PROGRAM PRG_LVCP5_Group1
VAR
    // Function Block Instance
    fbContactor: FB_ContactorControl;

    // Contactor 1 IO Structure  
    stContactor_IO: ST_ContactorIO;
    
    // Başlangıç konfigürasyonu için flag
    bContactorInitDone: BOOL := FALSE;
    bCapacitorInitDone: BOOL := FALSE;	
END_VAR



	M_Contactor();
	
	M_Capacitor();

METHOD M_Capacitor : BOOL
VAR
    nGroupIndex : INT;
END_VAR
	nGroupIndex := 0;  // Grup 1 için index
	
	IF NOT bCapacitorInitDone THEN
	
		// Grup 1 değerlerini ata
		GVL_LVCP5.astCompensationGroups[nGroupIndex].rPower := 10.0;
		GVL_LVCP5.astCompensationGroups[nGroupIndex].rVoltage := 450.0;
		GVL_LVCP5.astCompensationGroups[nGroupIndex].nQuantity := 10;
		GVL_LVCP5.astCompensationGroups[nGroupIndex].sTagPrefix := '+EP8-16C1';
		GVL_LVCP5.astCompensationGroups[nGroupIndex].sProductCode := 'ENT.CXD-450-10';
		
		bCapacitorInitDone := TRUE;
	END_IF
	
	// Grup 1 aktif durumu
	GVL_LVCP5.abGroupActive[nGroupIndex] := stContactor_IO.bFeedback;
	
	M_Capacitor := TRUE;
END_METHOD

METHOD M_Contactor : BOOL
VAR_INPUT
END_VAR
IF NOT bContactorInitDone THEN
    // Konfigürasyon parametreleri
    GVL_LVCP5.stGroup1_ContactorHMI.stConfig.sProjectCode := '+EP8-17K1';
    GVL_LVCP5.stGroup1_ContactorHMI.stConfig.sProductCode := 'SCH LC1G225LSEA';
    GVL_LVCP5.stGroup1_ContactorHMI.stConfig.rRatedCurrent := 225.0;
    GVL_LVCP5.stGroup1_ContactorHMI.stConfig.rRatedVoltage := 1000.0;
    GVL_LVCP5.stGroup1_ContactorHMI.stConfig.nPhaseCount := 3;
    GVL_LVCP5.stGroup1_ContactorHMI.stConfig.tFeedbackDelay := T#500MS;
    GVL_LVCP5.stGroup1_ContactorHMI.stConfig.tWeldedDelay := T#2S;
    GVL_LVCP5.stGroup1_ContactorHMI.stConfig.dwOperationLimit := 100000;
    
    // Başlangıç bakım sayacı
    GVL_LVCP5.stGroup1_ContactorHMI.stStatistics.dwRemainingOperations := GVL_LVCP5.stGroup1_ContactorHMI.stConfig.dwOperationLimit;
	
	bContactorInitDone := TRUE;
END_IF	
	
// Function Block Çağrısı
fbContactor(
    // Fiziksel Girişler
    bFeedback 		:= stContactor_IO.bFeedback,
    bPLCControl 	:= stContactor_IO.bPLCControl,
    
    // Güvenlik Girişleri
    bSafetyLoop 	:= GVL_Alarm.bSafetyLoop,
    bInterlock 		:= FALSE,
    
    // Sistem Girişleri
    bMasterReset 	:= GVL_Alarm.bMasterReset,
    
    // HMI Bağlantısı
    stHMI 			:= GVL_LVCP5.stGroup1_ContactorHMI,
    
    // Fiziksel Çıkış
    bOutput 		=> stContactor_IO.bOutput
);

// SQL Kayıt İşlemi
IF GVL_LVCP5.stGroup1_ContactorHMI.stStatistics.bNewOperationFlag THEN
    // SQL kayıt fonksiyonunu çağır
    GVL_LVCP5.stGroup1_ContactorHMI.stStatistics.bNewOperationFlag := FALSE;
END_IF
END_METHOD

END_PROGRAM

(* stored: Version 1.1.0.1, ProductVersion 3.1.4024.15
   POU PRG_LVCP5_Group1: Id {33f01a0b-2150-499b-9519-36de317c3bb8}, SpecialFunc None
   Method M_Capacitor: Id {48ceb8fd-ac5c-4ec2-bc2d-9fa6e52429f8}
   Method M_Contactor: Id {d611680a-d304-4d1b-889e-b4966053de2f} *)
